INTERFACE EventLogger

METHOD submit_event_message
VAR_INPUT
  ev: EventMessage;
END_VAR
END_METHOD

END_INTERFACE

(* stored: Version 1.1.0.1, ProductVersion 3.1.4024.9
   Itf EventLogger: Id {ed02ee8e-c48d-425b-b1ba-db2fe412fd83}
   Method submit_event_message: Id {f84ec892-41c2-4113-b29d-b2de8225110c} *)
